// TIA Portal V17 export
// export: Created 2023-12-05T13:40:23.9001439Z, ExportSetting WithDefaults, DisplayName Totally Integrated Automation Portal, DisplayVersion V17, DisplayName TIA Portal Openness, DisplayVersion V17, DisplayName TIA Portal Version Control Interface, DisplayVersion V17, DisplayName SINAMICS Startdrive Advanced, DisplayVersion V17, DisplayName SINAMICS Startdrive G130, G150, S120, S150, SINAMICS MV, S210, DisplayVersion V17, DisplayName SINAMICS Startdrive G110M, G120, G120C, G120D, G120P, G115D, DisplayVersion V17, DisplayName STEP 7 Professional, DisplayVersion V17, DisplayName STEP 7 Safety, DisplayVersion V17, DisplayName WinCC Professional, DisplayVersion V17
FUNCTION_BLOCK "FB400 Counters"   // FB400, LAD
{ S7_Optimized_Access := 'TRUE' }
VERSION : 0.1
// Block for counting OK/NOK/Doub/Total for 50 Version
// stored: AutoNumber false, IsIECCheckEnabled false, IsRetainMemResEnabled false, MemoryReserve 100, SetENOAutomatically false, UDAEnableTagReadback false
   VAR_INPUT
      Start : Bool;
      "Status OK" : Bool;
      "Status NOK" : Bool;
      "Staus Doub" : Bool;
      "One counter for machine" : Bool;
      "Version Nb" : Int;
   END_VAR
   VAR_IN_OUT
      "Reset Act" : Bool;
   END_VAR
   VAR
      St : Bool;
      Res : Bool;
      ResTot : Bool;
      Spare : Int;
   END_VAR
   VAR RETAIN
      Count { S7_SetPoint := 'True'} : "ProductionCounter";
   END_VAR
   VAR
      "Total OK" : DInt;
      "Total NOK" : DInt;
      "Total Doub" : DInt;
      "Total All" : DInt;
      "Act OK" : DInt;
      "Act NOK" : DInt;
      "Act Doub" : DInt;
      FP1 : Bool;
      FP2 : Bool;
   END_VAR
   VAR_TEMP
      zero : Int;
      ret : Int;
      i : Int;
   END_VAR
   // Count.V[1].Count.VersionOK := 1;
   // Count.V[2].Count.VersionOK := 2;
   // Count.V[3].Count.VersionOK := 3;
   // Count.V[4].Count.VersionOK := 4;
   // Count.V[5].Count.VersionOK := 5;
   // Count.V[6].Count.VersionOK := 6;
   // Count.V[7].Count.VersionOK := 7;
   // Count.V[8].Count.VersionOK := 8;
   // Count.V[9].Count.VersionOK := 9;
   // Count.V[10].Count.VersionOK := 10;
   // Count.V[11].Count.VersionOK := 11;
   // Count.V[12].Count.VersionOK := 12;
   // Count.V[13].Count.VersionOK := 13;
   // Count.V[14].Count.VersionOK := 14;
   // Count.V[15].Count.VersionOK := 15;
   // Count.V[16].Count.VersionOK := 16;
   // Count.V[17].Count.VersionOK := 17;
   // Count.V[18].Count.VersionOK := 18;
   // Count.V[19].Count.VersionOK := 19;
   // Count.V[20].Count.VersionOK := 20;
   // Count.V[21].Count.VersionOK := 21;
   // Count.V[22].Count.VersionOK := 22;
   // Count.V[23].Count.VersionOK := 23;
   // Count.V[24].Count.VersionOK := 24;
   // Count.V[25].Count.VersionOK := 25;
   // Count.V[26].Count.VersionOK := 26;
   // Count.V[27].Count.VersionOK := 27;
   // Count.V[28].Count.VersionOK := 28;
   // Count.V[29].Count.VersionOK := 29;
   // Count.V[30].Count.VersionOK := 30;
   // Count.V[1].Count.VersionNOK := 1;
   // Count.V[2].Count.VersionNOK := 2;
   // Count.V[3].Count.VersionNOK := 3;
   // Count.V[4].Count.VersionNOK := 4;
   // Count.V[5].Count.VersionNOK := 5;
   // Count.V[6].Count.VersionNOK := 6;
   // Count.V[7].Count.VersionNOK := 7;
   // Count.V[8].Count.VersionNOK := 8;
   // Count.V[9].Count.VersionNOK := 9;
   // Count.V[10].Count.VersionNOK := 10;
   // Count.V[11].Count.VersionNOK := 11;
   // Count.V[12].Count.VersionNOK := 12;
   // Count.V[13].Count.VersionNOK := 13;
   // Count.V[14].Count.VersionNOK := 14;
   // Count.V[15].Count.VersionNOK := 15;
   // Count.V[16].Count.VersionNOK := 16;
   // Count.V[17].Count.VersionNOK := 17;
   // Count.V[18].Count.VersionNOK := 18;
   // Count.V[19].Count.VersionNOK := 19;
   // Count.V[20].Count.VersionNOK := 20;
   // Count.V[21].Count.VersionNOK := 21;
   // Count.V[22].Count.VersionNOK := 22;
   // Count.V[23].Count.VersionNOK := 23;
   // Count.V[24].Count.VersionNOK := 24;
   // Count.V[25].Count.VersionNOK := 25;
   // Count.V[26].Count.VersionNOK := 26;
   // Count.V[27].Count.VersionNOK := 27;
   // Count.V[28].Count.VersionNOK := 28;
   // Count.V[29].Count.VersionNOK := 29;
   // Count.V[30].Count.VersionNOK := 30;
   // Count.V[1].Count.VersionDoub := 1;
   // Count.V[2].Count.VersionDoub := 2;
   // Count.V[3].Count.VersionDoub := 3;
   // Count.V[4].Count.VersionDoub := 4;
   // Count.V[5].Count.VersionDoub := 5;
   // Count.V[6].Count.VersionDoub := 6;
   // Count.V[7].Count.VersionDoub := 7;
   // Count.V[8].Count.VersionDoub := 8;
   // Count.V[9].Count.VersionDoub := 9;
   // Count.V[10].Count.VersionDoub := 10;
   // Count.V[11].Count.VersionDoub := 11;
   // Count.V[12].Count.VersionDoub := 12;
   // Count.V[13].Count.VersionDoub := 13;
   // Count.V[14].Count.VersionDoub := 14;
   // Count.V[15].Count.VersionDoub := 15;
   // Count.V[16].Count.VersionDoub := 16;
   // Count.V[17].Count.VersionDoub := 17;
   // Count.V[18].Count.VersionDoub := 18;
   // Count.V[19].Count.VersionDoub := 19;
   // Count.V[20].Count.VersionDoub := 20;
   // Count.V[21].Count.VersionDoub := 21;
   // Count.V[22].Count.VersionDoub := 22;
   // Count.V[23].Count.VersionDoub := 23;
   // Count.V[24].Count.VersionDoub := 24;
   // Count.V[25].Count.VersionDoub := 25;
   // Count.V[26].Count.VersionDoub := 26;
   // Count.V[27].Count.VersionDoub := 27;
   // Count.V[28].Count.VersionDoub := 28;
   // Count.V[29].Count.VersionDoub := 29;
   // Count.V[30].Count.VersionDoub := 30;
   // Count.V[1].Count.TotalOK := 1;
   // Count.V[2].Count.TotalOK := 2;
   // Count.V[3].Count.TotalOK := 3;
   // Count.V[4].Count.TotalOK := 4;
   // Count.V[5].Count.TotalOK := 5;
   // Count.V[6].Count.TotalOK := 6;
   // Count.V[7].Count.TotalOK := 7;
   // Count.V[8].Count.TotalOK := 8;
   // Count.V[9].Count.TotalOK := 9;
   // Count.V[10].Count.TotalOK := 10;
   // Count.V[11].Count.TotalOK := 11;
   // Count.V[12].Count.TotalOK := 12;
   // Count.V[13].Count.TotalOK := 13;
   // Count.V[14].Count.TotalOK := 14;
   // Count.V[15].Count.TotalOK := 15;
   // Count.V[16].Count.TotalOK := 16;
   // Count.V[17].Count.TotalOK := 17;
   // Count.V[18].Count.TotalOK := 18;
   // Count.V[19].Count.TotalOK := 19;
   // Count.V[20].Count.TotalOK := 20;
   // Count.V[21].Count.TotalOK := 21;
   // Count.V[22].Count.TotalOK := 22;
   // Count.V[23].Count.TotalOK := 23;
   // Count.V[24].Count.TotalOK := 24;
   // Count.V[25].Count.TotalOK := 25;
   // Count.V[26].Count.TotalOK := 26;
   // Count.V[27].Count.TotalOK := 27;
   // Count.V[28].Count.TotalOK := 28;
   // Count.V[29].Count.TotalOK := 29;
   // Count.V[30].Count.TotalOK := 30;
   // Count.V[1].Count.TotalNOK := 1;
   // Count.V[2].Count.TotalNOK := 2;
   // Count.V[3].Count.TotalNOK := 3;
   // Count.V[4].Count.TotalNOK := 4;
   // Count.V[5].Count.TotalNOK := 5;
   // Count.V[6].Count.TotalNOK := 6;
   // Count.V[7].Count.TotalNOK := 7;
   // Count.V[8].Count.TotalNOK := 8;
   // Count.V[9].Count.TotalNOK := 9;
   // Count.V[10].Count.TotalNOK := 10;
   // Count.V[11].Count.TotalNOK := 11;
   // Count.V[12].Count.TotalNOK := 12;
   // Count.V[13].Count.TotalNOK := 13;
   // Count.V[14].Count.TotalNOK := 14;
   // Count.V[15].Count.TotalNOK := 15;
   // Count.V[16].Count.TotalNOK := 16;
   // Count.V[17].Count.TotalNOK := 17;
   // Count.V[18].Count.TotalNOK := 18;
   // Count.V[19].Count.TotalNOK := 19;
   // Count.V[20].Count.TotalNOK := 20;
   // Count.V[21].Count.TotalNOK := 21;
   // Count.V[22].Count.TotalNOK := 22;
   // Count.V[23].Count.TotalNOK := 23;
   // Count.V[24].Count.TotalNOK := 24;
   // Count.V[25].Count.TotalNOK := 25;
   // Count.V[26].Count.TotalNOK := 26;
   // Count.V[27].Count.TotalNOK := 27;
   // Count.V[28].Count.TotalNOK := 28;
   // Count.V[29].Count.TotalNOK := 29;
   // Count.V[30].Count.TotalNOK := 30;
   // Count.V[1].Count.TotalDoub := 1;
   // Count.V[2].Count.TotalDoub := 2;
   // Count.V[3].Count.TotalDoub := 3;
   // Count.V[4].Count.TotalDoub := 4;
   // Count.V[5].Count.TotalDoub := 5;
   // Count.V[6].Count.TotalDoub := 6;
   // Count.V[7].Count.TotalDoub := 7;
   // Count.V[8].Count.TotalDoub := 8;
   // Count.V[9].Count.TotalDoub := 9;
   // Count.V[10].Count.TotalDoub := 10;
   // Count.V[11].Count.TotalDoub := 11;
   // Count.V[12].Count.TotalDoub := 12;
   // Count.V[13].Count.TotalDoub := 13;
   // Count.V[14].Count.TotalDoub := 14;
   // Count.V[15].Count.TotalDoub := 15;
   // Count.V[16].Count.TotalDoub := 16;
   // Count.V[17].Count.TotalDoub := 17;
   // Count.V[18].Count.TotalDoub := 18;
   // Count.V[19].Count.TotalDoub := 19;
   // Count.V[20].Count.TotalDoub := 20;
   // Count.V[21].Count.TotalDoub := 21;
   // Count.V[22].Count.TotalDoub := 22;
   // Count.V[23].Count.TotalDoub := 23;
   // Count.V[24].Count.TotalDoub := 24;
   // Count.V[25].Count.TotalDoub := 25;
   // Count.V[26].Count.TotalDoub := 26;
   // Count.V[27].Count.TotalDoub := 27;
   // Count.V[28].Count.TotalDoub := 28;
   // Count.V[29].Count.TotalDoub := 29;
   // Count.V[30].Count.TotalDoub := 30;
   VAR_TEMP   // added for the SCL form of the ladder/FBD networks
      _w1 : Bool;
   END_VAR
BEGIN

REGION Network 1: Start
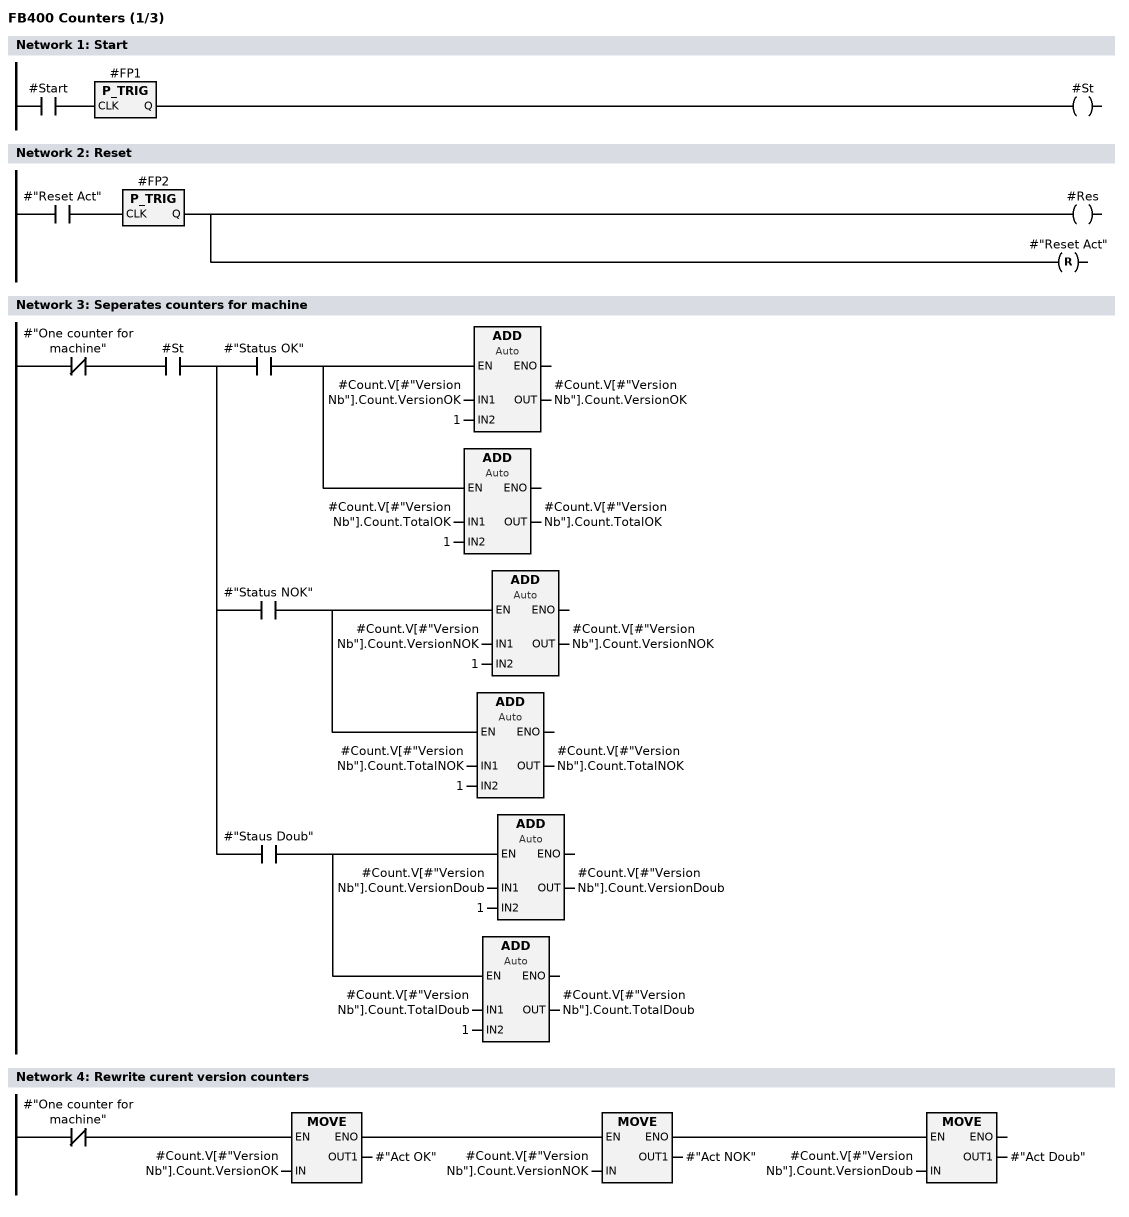
   RUNG wire#powerrail
      Contact( #Start )
      P_Trig( #FP1 )
      Coil( #St )
   END_RUNG
   // the same network as SCL:
   #_w1 := #Start AND NOT #FP1;   // rising edge
   #FP1 := #Start;
   #St := #_w1;
END_REGION

REGION Network 2: Reset
   RUNG wire#powerrail
      Contact( #"Reset Act" )
      P_Trig( #FP2 )
      wire#w1
      Coil( #Res )
   END_RUNG
   RUNG wire#w1
      R_Coil( #"Reset Act" )
   END_RUNG
   // the same network as SCL:
   #_w1 := #"Reset Act" AND NOT #FP2;   // rising edge
   #FP2 := #"Reset Act";
   #Res := #_w1;
   IF #_w1 THEN #"Reset Act" := FALSE; END_IF;
END_REGION

REGION Network 3: Seperates counters for machine
   RUNG wire#powerrail
      I_Contact( #"One counter for machine" )
      Contact( #St )
      wire#w1
      Contact( #"Status OK" )
      wire#w2
      Add(in1 := #Count.V[#"Version Nb"].Count.VersionOK, in2 := 1, out => #Count.V[#"Version Nb"].Count.VersionOK)
   END_RUNG
   RUNG wire#w2
      Add(in1 := #Count.V[#"Version Nb"].Count.TotalOK, in2 := 1, out => #Count.V[#"Version Nb"].Count.TotalOK)
   END_RUNG
   RUNG wire#w1
      Contact( #"Status NOK" )
      wire#w3
      Add(in1 := #Count.V[#"Version Nb"].Count.VersionNOK, in2 := 1, out => #Count.V[#"Version Nb"].Count.VersionNOK)
   END_RUNG
   RUNG wire#w3
      Add(in1 := #Count.V[#"Version Nb"].Count.TotalNOK, in2 := 1, out => #Count.V[#"Version Nb"].Count.TotalNOK)
   END_RUNG
   RUNG wire#w1
      Contact( #"Staus Doub" )
      wire#w4
      Add(in1 := #Count.V[#"Version Nb"].Count.VersionDoub, in2 := 1, out => #Count.V[#"Version Nb"].Count.VersionDoub)
   END_RUNG
   RUNG wire#w4
      Add(in1 := #Count.V[#"Version Nb"].Count.TotalDoub, in2 := 1, out => #Count.V[#"Version Nb"].Count.TotalDoub)
   END_RUNG
   // the same network as SCL:
   #_w1 := NOT #"One counter for machine" AND #St;
   IF #_w1 AND #"Status OK" THEN
       #Count.V[#"Version Nb"].Count.VersionOK := #Count.V[#"Version Nb"].Count.VersionOK + 1;
       #Count.V[#"Version Nb"].Count.TotalOK := #Count.V[#"Version Nb"].Count.TotalOK + 1;
   END_IF;
   IF #_w1 AND #"Status NOK" THEN
       #Count.V[#"Version Nb"].Count.VersionNOK := #Count.V[#"Version Nb"].Count.VersionNOK + 1;
       #Count.V[#"Version Nb"].Count.TotalNOK := #Count.V[#"Version Nb"].Count.TotalNOK + 1;
   END_IF;
   IF #_w1 AND #"Staus Doub" THEN
       #Count.V[#"Version Nb"].Count.VersionDoub := #Count.V[#"Version Nb"].Count.VersionDoub + 1;
       #Count.V[#"Version Nb"].Count.TotalDoub := #Count.V[#"Version Nb"].Count.TotalDoub + 1;
   END_IF;
END_REGION

REGION Network 4: Rewrite curent version counters
   RUNG wire#powerrail
      I_Contact( #"One counter for machine" )
      Move(in := #Count.V[#"Version Nb"].Count.VersionOK, out1 => #"Act OK")
      Move(in := #Count.V[#"Version Nb"].Count.VersionNOK, out1 => #"Act NOK")
      Move(in := #Count.V[#"Version Nb"].Count.VersionDoub, out1 => #"Act Doub")
   END_RUNG
   // the same network as SCL:
   IF NOT #"One counter for machine" THEN
       #"Act OK" := #Count.V[#"Version Nb"].Count.VersionOK;
       #"Act NOK" := #Count.V[#"Version Nb"].Count.VersionNOK;
       #"Act Doub" := #Count.V[#"Version Nb"].Count.VersionDoub;
   END_IF;
END_REGION

REGION Network 5: One counter for machine
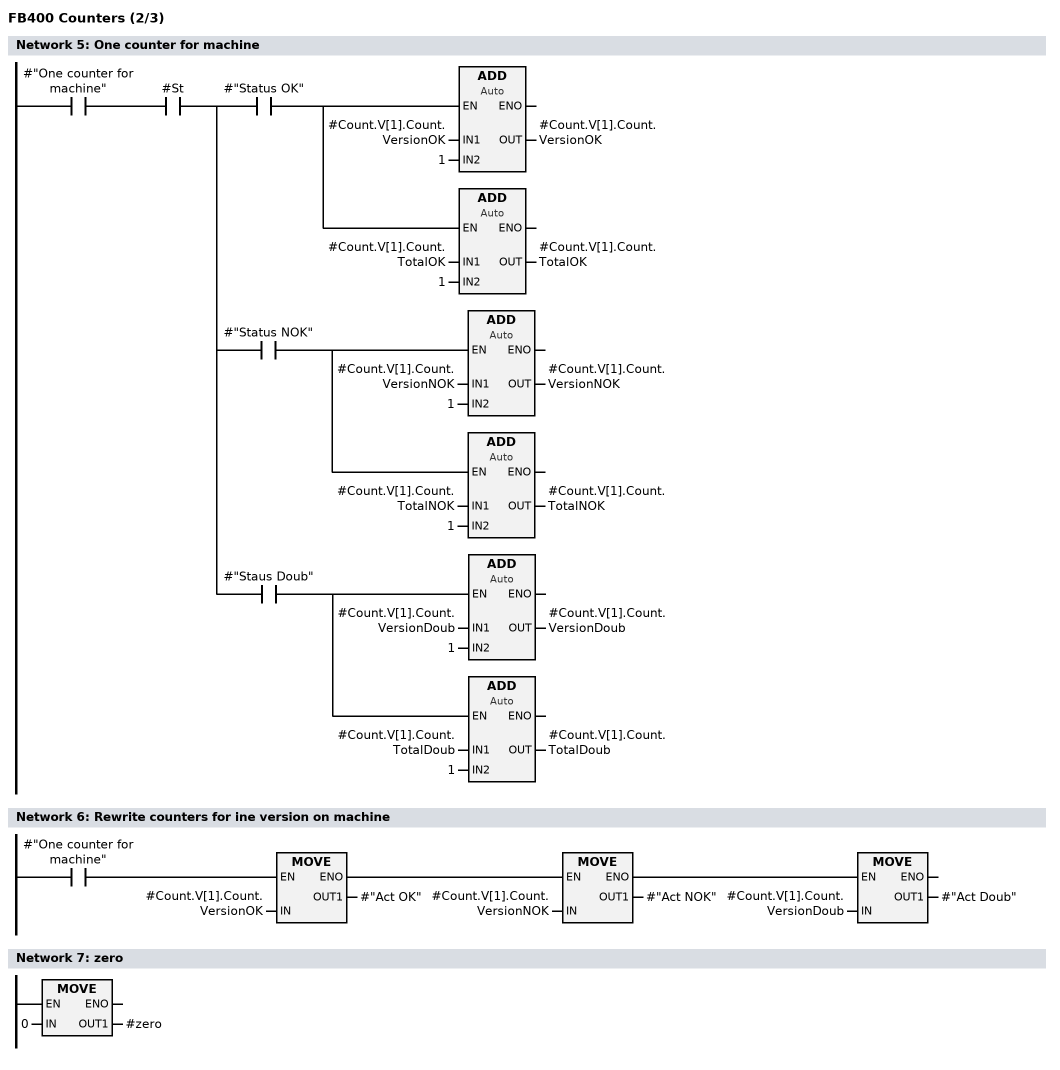
   RUNG wire#powerrail
      Contact( #"One counter for machine" )
      Contact( #St )
      wire#w1
      Contact( #"Status OK" )
      wire#w2
      Add(in1 := #Count.V[1].Count.VersionOK, in2 := 1, out => #Count.V[1].Count.VersionOK)
   END_RUNG
   RUNG wire#w2
      Add(in1 := #Count.V[1].Count.TotalOK, in2 := 1, out => #Count.V[1].Count.TotalOK)
   END_RUNG
   RUNG wire#w1
      Contact( #"Status NOK" )
      wire#w3
      Add(in1 := #Count.V[1].Count.VersionNOK, in2 := 1, out => #Count.V[1].Count.VersionNOK)
   END_RUNG
   RUNG wire#w3
      Add(in1 := #Count.V[1].Count.TotalNOK, in2 := 1, out => #Count.V[1].Count.TotalNOK)
   END_RUNG
   RUNG wire#w1
      Contact( #"Staus Doub" )
      wire#w4
      Add(in1 := #Count.V[1].Count.VersionDoub, in2 := 1, out => #Count.V[1].Count.VersionDoub)
   END_RUNG
   RUNG wire#w4
      Add(in1 := #Count.V[1].Count.TotalDoub, in2 := 1, out => #Count.V[1].Count.TotalDoub)
   END_RUNG
   // the same network as SCL:
   #_w1 := #"One counter for machine" AND #St;
   IF #_w1 AND #"Status OK" THEN
       #Count.V[1].Count.VersionOK := #Count.V[1].Count.VersionOK + 1;
       #Count.V[1].Count.TotalOK := #Count.V[1].Count.TotalOK + 1;
   END_IF;
   IF #_w1 AND #"Status NOK" THEN
       #Count.V[1].Count.VersionNOK := #Count.V[1].Count.VersionNOK + 1;
       #Count.V[1].Count.TotalNOK := #Count.V[1].Count.TotalNOK + 1;
   END_IF;
   IF #_w1 AND #"Staus Doub" THEN
       #Count.V[1].Count.VersionDoub := #Count.V[1].Count.VersionDoub + 1;
       #Count.V[1].Count.TotalDoub := #Count.V[1].Count.TotalDoub + 1;
   END_IF;
END_REGION

REGION Network 6: Rewrite counters for ine version on machine
   RUNG wire#powerrail
      Contact( #"One counter for machine" )
      Move(in := #Count.V[1].Count.VersionOK, out1 => #"Act OK")
      Move(in := #Count.V[1].Count.VersionNOK, out1 => #"Act NOK")
      Move(in := #Count.V[1].Count.VersionDoub, out1 => #"Act Doub")
   END_RUNG
   // the same network as SCL:
   IF #"One counter for machine" THEN
       #"Act OK" := #Count.V[1].Count.VersionOK;
       #"Act NOK" := #Count.V[1].Count.VersionNOK;
       #"Act Doub" := #Count.V[1].Count.VersionDoub;
   END_IF;
END_REGION

REGION Network 7: zero
   RUNG wire#powerrail
      Move(in := 0, out1 => #zero)
   END_RUNG
   // the same network as SCL:
   #zero := 0;
END_REGION

REGION Network 8: Fill zero to counters
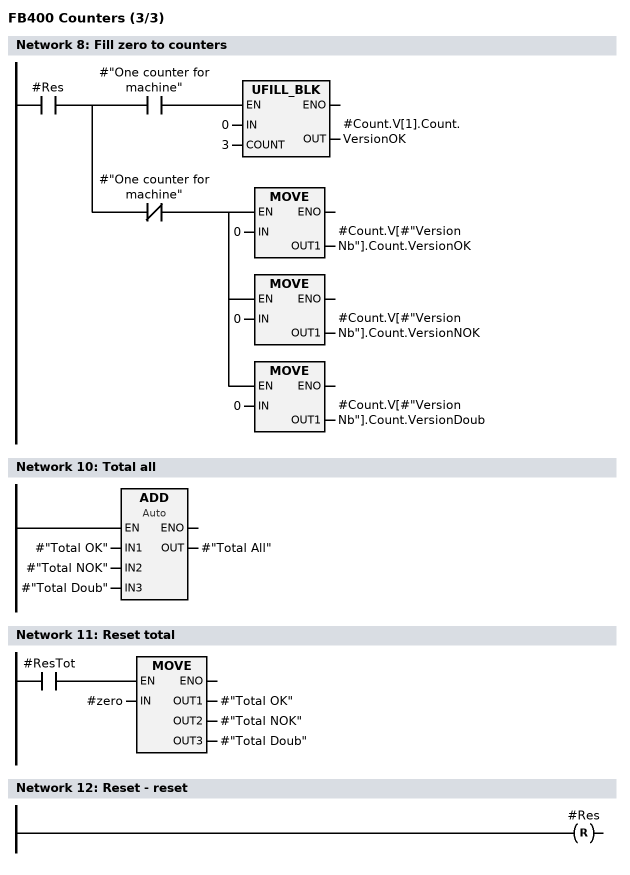
   IF #Res AND #"One counter for machine" THEN
       UFILL_BLK(IN := 0, COUNT := 3, OUT => #Count.V[1].Count.VersionOK);
   END_IF;
   IF #Res AND NOT #"One counter for machine" THEN
       #Count.V[#"Version Nb"].Count.VersionOK := 0;
       #Count.V[#"Version Nb"].Count.VersionNOK := 0;
       #Count.V[#"Version Nb"].Count.VersionDoub := 0;
   END_IF;
END_REGION

REGION Network 9 (SCL): Reset actual counters
   IF #Res THEN
       FOR #i := 1 TO 50 BY 1 DO
           #Count.V[#i].Count.VersionOK := 0;
           #Count.V[#i].Count.VersionNOK := 0;
           #Count.V[#i].Count.VersionDoub := 0;
       END_FOR;
   END_IF;
END_REGION

REGION Network 10: Total all
   RUNG wire#powerrail
      Add(in1 := #"Total OK", in2 := #"Total NOK", in3 := #"Total Doub", out => #"Total All")
   END_RUNG
   // the same network as SCL:
   #"Total All" := #"Total OK" + #"Total NOK" + #"Total Doub";
END_REGION

REGION Network 11: Reset total
   RUNG wire#powerrail
      Contact( #ResTot )
      Move(in := #zero, out1 => #"Total OK", out2 => #"Total NOK", out3 => #"Total Doub")
   END_RUNG
   // the same network as SCL:
   IF #ResTot THEN
       #"Total OK" := #zero;
       #"Total NOK" := #zero;
       #"Total Doub" := #zero;
   END_IF;
END_REGION

REGION Network 12: Reset - reset
   RUNG wire#powerrail
      R_Coil( #Res )
   END_RUNG
   // the same network as SCL:
   #Res := FALSE;
END_REGION
END_FUNCTION_BLOCK
